VAR_GLOBAL
//	GAB_FactoryIO_Inputs : ARRAY [0..1] OF WORD;
//	GAB_FactoryIO_InputRegs : ARRAY [0..7] OF INT;
//	GAB_FactoryIO_Outputs : ARRAY [0..1] OF WORD;
//	GAB_FactoryIO_OutputsRegs : ARRAY [0..7] OF INT;
END_VAR

(* stored: Version 1.1.0.1, ProductVersion 3.1.4024.11
   GVL GVL_FactoryIO_WebSample: Id {ae52c57a-5705-4df6-9b9e-cd21c7bcba13} *)
